Staubli VAL3: getStatus.pgx

public program getStatus(bool& x_bStatus[], string x_sItem)
  local num l_nSize
begin
  // give back the status
  x_bStatus=saveInOut:dInput[x_sItem].dDio
end
